PROGRAM Task_2
VAR
	tmrElevatorMove : TON;                  // Timer for the elevator movement
    bLocalAccessGranted : BOOL := FALSE;    // Local copy of the access granted status
    bLocalElevatorRequest : BOOL := FALSE;  // Local copy of the elevator request status
END_VAR

// Read the GVL variables locally to ensure correct types
bLocalAccessGranted := GVL.bAccessGranted;
bLocalElevatorRequest := GVL.bElevatorRequest;

// Elevator control logic
IF bLocalAccessGranted AND bLocalElevatorRequest THEN
    tmrElevatorMove(IN := TRUE, PT := GVL.tElevatorMoveTime);   // Start the elevator movement timer
ELSE
    tmrElevatorMove(IN := FALSE);
END_IF

// Update elevator status in the GVL
IF tmrElevatorMove.Q THEN
    GVL.bElevatorArrived := TRUE;     // Set TRUE when elevator arrives at floor 0
ELSE
    GVL.bElevatorArrived := FALSE;
END_IF

END_PROGRAM

(* stored: Version 1.1.0.1, ProductVersion 3.1.4024.12
   POU Task_2: Id {f622ca62-79f6-4411-bbe8-a47044c7fd49}, SpecialFunc None *)
